# EPICS substitutions: scllrfApp/Db/BuncherWFtoGunWF.substitutions
file BuncherWFtoGunWF.template
{
{PRC1=100:PRL,PRC2=100:PRC:SPARE1,PRC3=100:PRC:SPARE2,PRC4=100:CAV1,PRC5=100:CAV2,PRC6=100:PRC:SPARE3,PRC7=100:PRC:SPARE4,PRC8=100:LASR,PRC9=100:PRC:SPARE5,PRC10=100:PRC:SPARE6,PRC11=100:PRC:SPARE7,PRC12=100:PRC:SPARE8,PRC13=100:PRC:SPARE9,PRC14=100:PRC:SPARE10,PRC15=100:PRC:SPARE11,PRC16=100:PRC:SPARE12,RFS11=100:DRV1,RFS12=100:DRV1A,RFS13=S100:FWD1,RFS14=S100:REV1,RFS15=100:FWD1,RFS16=100:REV1,RFS17=C100:FWD1,RFS18=C100:REV1,RFS19=100:RFS1:SPARE1,RFS110=100:RFS1:DAC,RFS111=100:RFS1:SPARE2,RFS112=100:RFS1:SPARE3,RFS113=100:RFS1:SPARE4,RFS114=100:RFS1:SPARE5,RFS115=100:RFS1:SPARE6,RFS116=100:RFS1:SPARE7,RFS21=100:DRV2,RFS22=100:DRV2A,RFS23=S100:FWD2,RFS24=S100:REV2,RFS25=100:FWD2,RFS26=100:REV2,RFS27=C100:FWD2,RFS28=C100:REV2,RFS29=100:RFS2:SPARE1,RFS210=100:RFS2:DAC,RFS211=100:RFS2:SPARE2,RFS212=100:RFS2:SPARE3,RFS213=100:RFS2:SPARE4,RFS214=100:RFS2:SPARE5,RFS215=100:RFS2:SPARE6,RFS215=100:RFS2:SPARE7}
}
